Yaskawa INFORM job: BUTTERFLY.JBI

/JOB
//NAME BUTTERFLY
//POS
///NPOS 22,0,0,0,0,0
///TOOL 0
///POSTYPE PULSE
///PULSE
C00000=-2822,58859,-1118,-1041,-34109,-89
C00001=-2153,58790,-1248,-1130,-34038,-357
C00002=-2415,58500,-1692,-1101,-33859,-248
C00003=-2588,58146,-2230,-1083,-33643,-174
C00004=-2715,58309,-1987,-1064,-33742,-125
C00005=-2865,58359,-1913,-1044,-33771,-65
C00006=-2782,57960,-2513,-1060,-33531,-94
C00007=-2802,57835,-2702,-1060,-33455,-84
C00008=-2740,57486,-3228,-1073,-33243,-105
C00009=-2595,57124,-3774,-1098,-33023,-159
C00010=-2411,56761,-4321,-1128,-32801,-228
C00011=-2117,56486,-4737,-1172,-32630,-341
C00012=-1932,56652,-4486,-1195,-32730,-417
C00013=-1549,56488,-4735,-1249,-32625,-568
C00014=-1126,56501,-4715,-1306,-32628,-737
C00015=-1077,56886,-4127,-1306,-32867,-762
C00016=-1229,57257,-3562,-1278,-33098,-707
C00017=-1456,57604,-3036,-1242,-33313,-621
C00018=-1477,57989,-2450,-1232,-33550,-618
C00019=-1517,58384,-1850,-1220,-33793,-607
C00020=-1849,58549,-1606,-1174,-33893,-476
C00021=-2153,58790,-1248,-1130,-34038,-357
//INST
///DATE 2026/04/15 15:34
///ATTR SC,RW
///GROUP1 RB1
NOP
MOVJ C00000 VJ=0.78
MOVJ C00001 VJ=0.78
MOVJ C00002 VJ=0.78
MOVJ C00003 VJ=0.78
MOVJ C00004 VJ=0.78
MOVJ C00005 VJ=0.78
MOVJ C00006 VJ=0.78
MOVJ C00007 VJ=0.78
MOVJ C00008 VJ=0.78
MOVJ C00009 VJ=0.78
MOVJ C00010 VJ=0.78
MOVJ C00011 VJ=0.78
MOVJ C00012 VJ=0.78
MOVJ C00013 VJ=0.78
MOVJ C00014 VJ=0.78
MOVJ C00015 VJ=0.78
MOVJ C00016 VJ=0.78
MOVJ C00017 VJ=0.78
MOVJ C00018 VJ=0.78
MOVJ C00019 VJ=0.78
MOVJ C00020 VJ=0.78
MOVJ C00021 VJ=0.78
END
